ABB RobotStudio station: Lab3.rsstnx

Station Lab3 (saved by RobotStudio 24.3.10885.0)
Layout (positions relative to the parent item):
